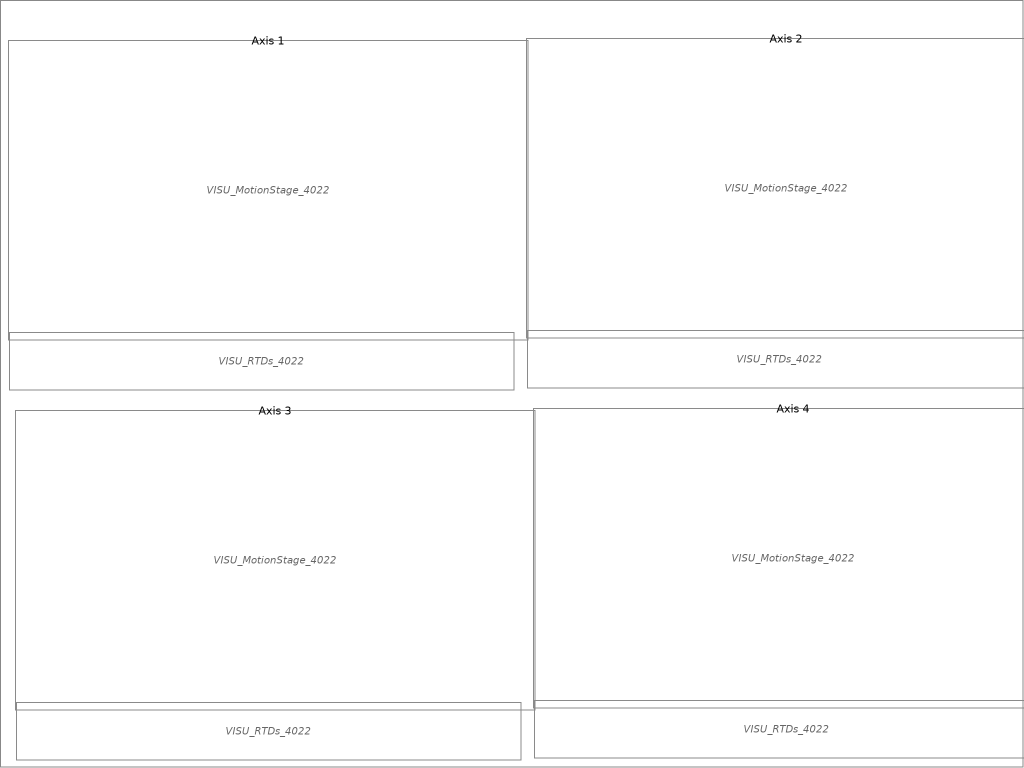
VISUALIZATION AT2K2_4022  // 1024x768
    Frame (8,40 520x300)
        shows VISU_MotionStage_4022(VisuMotionStage := Main.M1, Extras := PRG_2_AT1K4.fbStage1.stExtra)
    Label (193,26 150x30), "Axis 1"
    Frame (9,332 505x58)
        shows VISU_RTDs_4022(fTemp1 := PRG_2_AT1K4.fbStage1.fTemp1, fTemp2 := PRG_2_AT1K4.fbStage1.fTemp2)
    Frame (526,38 520x300)
        shows VISU_MotionStage_4022(VisuMotionStage := Main.M2, Extras := PRG_2_AT1K4.fbStage2.stExtra)
    Label (711,24 150x30), "Axis 2"
    Frame (527,330 505x58)
        shows VISU_RTDs_4022(fTemp1 := PRG_2_AT1K4.fbStage2.fTemp1, fTemp2 := PRG_2_AT1K4.fbStage2.fTemp2)
    Frame (15,410 520x300)
        shows VISU_MotionStage_4022(VisuMotionStage := Main.M3, Extras := PRG_2_AT1K4.fbStage3.stExtra)
    Label (200,396 150x30), "Axis 3"
    Frame (16,702 505x58)
        shows VISU_RTDs_4022(fTemp1 := PRG_2_AT1K4.fbStage3.fTemp1, fTemp2 := PRG_2_AT1K4.fbStage3.fTemp2)
    Frame (533,408 520x300)
        shows VISU_MotionStage_4022(VisuMotionStage := Main.M4, Extras := PRG_2_AT1K4.fbStage4.stExtra)
    Label (718,394 150x30), "Axis 4"
    Frame (534,700 505x58)
        shows VISU_RTDs_4022(fTemp1 := PRG_2_AT1K4.fbStage4.fTemp1, fTemp2 := PRG_2_AT1K4.fbStage4.fTemp2)
END_VISUALIZATION

(* stored: Version 1.1.0.1, ProductVersion 3.1.4022.18
   Visu AT2K2_4022: Id {de500e0a-39e0-4007-92a3-02ecc8a61697} *)
